// TIA Portal V16 export
// export: Created 2024-12-03T15:41:42.9786979Z, ExportSetting WithDefaults, DisplayName Totally Integrated Automation Portal, DisplayVersion V16 Update 6, DisplayName TIA Portal Version Control Interface, DisplayVersion V16 Update 2, DisplayName TIA Portal Openness, DisplayVersion V16 Update 6, DisplayName TIA Portal Teamcenter Gateway, DisplayVersion V16, DisplayName SINAMICS Startdrive Advanced, DisplayVersion V16 Update 5, DisplayName SINAMICS Startdrive G130, G150, S120, S150, SINAMICS MV, S210, DisplayVersion V16 Update 5, DisplayName SINAMICS Startdrive G110M, G120, G120C, G120D, G120P, G115D, DisplayVersion V16 Update 5, DisplayName STEP 7 Professional, DisplayVersion V16 Update 6, DisplayName STEP 7 Safety, DisplayVersion V16, DisplayName WinCC Advanced / Unified PC, DisplayVersion V16 Update 6
FUNCTION_BLOCK "ZPA_Controller"   // FB23, SCL
{ S7_Optimized_Access := 'TRUE' }
VERSION : 0.1
// stored: AutoNumber true, IsIECCheckEnabled false, IsRetainMemResEnabled false, MemoryReserve 100, SetENOAutomatically false, UDAEnableTagReadback false
   VAR_INPUT
      I_ConnectUpStream : Bool := TRUE;
      I_StartedAutoMode : Bool;
      I_UseEncoder : Bool := true;
      I_BuildName : Bool := true;
      I_UseExternalReset : Bool := TRUE;
   END_VAR
   VAR_IN_OUT
      IO_Upstream : "Conveyor_UDT";
      IO_DownStream : "Conveyor_UDT";
      IO_COnv : "Conveyor_UDT";
   END_VAR
   VAR
      cyclerun : "CycleRun";
      Alarm : "AlarmInfo_UDT";
      AlarmInfoValue : String;
      ConveyorMode : Int;
      StepNumber : DInt;
      PrevStepNumber : DInt;
      ObjectRequestedMemory : Bool;
      ObjectReceivedFromDownStream : Bool;
      Step_105_GapTimeOk : Bool;
      GapTimeTimer : "TON_Encoder_FB";
      SleepTimer { S7_SetPoint := 'True'} : "TON_Encoder_FB";
      ToCloseDetection { S7_SetPoint := 'True'} : "TON_Encoder_FB";
      ToLongDetectionEnd { S7_SetPoint := 'True'} : "TON_Encoder_FB";
      ToLongDetectionStart { S7_SetPoint := 'True'} : "TON_Encoder_FB";
      ToSmallDetection { S7_SetPoint := 'True'} : "TON_Encoder_FB";
      DownStreamIsRunning { S7_SetPoint := 'True'} : Bool;
      DownStreamRunningPredictor : Int;
      ObjectReceivedDuringSending : Bool;
      BlockedRetry : Int;
      InitializeInternal : Bool;
      diag : Struct
         TrackingLost : UInt;
      END_STRUCT;
      StartupDelay : TON_TIME;
      Step_Init_10 { S7_SetPoint := 'True'} : "StepperController_Encoder";
      Step_Send_WaitAccumulate_100 { S7_SetPoint := 'True'} : "StepperController_Encoder";
      Step_Send_WaitReceive_105 { S7_SetPoint := 'True'} : "StepperController_Encoder";
      Step_Send_Sending_110 { S7_SetPoint := 'True'} : "StepperController_Encoder";
      Step_Send_RunEmpty_120 { S7_SetPoint := 'True'} : "StepperController_Encoder";
      Step_Rec_Waiting_200 { S7_SetPoint := 'True'} : "StepperController";
      Step_Rec_Request_210 { S7_SetPoint := 'True'} : "StepperController_Encoder";
      Step_Rec_receivingTillEnd_215 { S7_SetPoint := 'True'} : "StepperController_Encoder";
      Step_Rec_RequetContiue_220 { S7_SetPoint := 'True'} : "StepperController_Encoder";
      Step_RequestObject_400_1 { S7_SetPoint := 'True'} : "StepperController_Encoder";
      Step_RequestObject_400_2 { S7_SetPoint := 'True'} : "StepperController_Encoder";
      Encoder { S7_SetPoint := 'True'} : "Virtual_Encoder_FB";
      BlockAlarmReceive { S7_SetPoint := 'True'} : Program_Alarm;
      BlockedSending { S7_SetPoint := 'True'} : Program_Alarm;
      ToCloseALarm { S7_SetPoint := 'True'} : Program_Alarm;
      ToSmallAlarm { S7_SetPoint := 'True'} : Program_Alarm;
      ToLongAlarm { S7_SetPoint := 'True'} : Program_Alarm;
      ResetMirror { S7_SetPoint := 'True'} : Bool;
   END_VAR
   VAR_TEMP
      T_ZoneInfo : "ZoneInfo";
      T_Appstate : "ApplicationState_UDT";
      T_Condition : Bool;
      T_Condtion_1 : Bool;
      T_Condtion_2 : Bool;
      T_NextStepNumber : DInt;
      T_TimeOutStepNumber : DInt;
      T_ConditionTime : Time;
      T_RunSent : Bool;
      T_RunReceive : Bool;
      T_RunInit : Bool;
      T_ReceiveTransferUnit : Bool;
      T_SleepMode : Bool;
      T_StandbyMode : Bool;
      T_Dummy : Bool;
   END_VAR
   VAR CONSTANT
      Step_TimeOutSending : DInt := 910;
      Step_TImeOutReceiving : DInt := 810;
      Step_ToCloseAlarm : DInt := 920;
      Step_ToSmall : DInt := 930;
      Step_ToLong : DInt := 940;
   END_VAR
BEGIN
   #T_ZoneInfo := "ApplicationState_DB".ZoneNames[#IO_COnv.Zone];
   #T_Appstate := "ApplicationState_DB".Appstate[#T_ZoneInfo.AppStateIndex];
   #ConveyorMode := #IO_COnv.Settings.Mode;

   IF "RunTime_DB".CycleRun = #T_ZoneInfo.AppStateIndex THEN
       #cyclerun();
   END_IF;

   #T_NextStepNumber := 0;
   #T_Condition := false;

   REGION ENCODER

       IF #I_UseEncoder THEN

           IF #IO_COnv.Cmd.RunAuto AND #IO_COnv.Input.Running_FB THEN
               #Encoder.I_CurrentRelativeSpeed_Perc := #IO_COnv.Cmd.SpeedAuto;
           ELSE
               #Encoder.I_CurrentRelativeSpeed_Perc := 0.0;
           END_IF;

           #Encoder(I_RelativeReferenceSpeed_Perc := #IO_COnv.Encoder.Settings.BaseRelative,
                    I_AbsoluteSpeedOnReferecne_m_min := #IO_COnv.Encoder.Settings.Base_M_min,
                    IO_VirtualEncoder := #IO_COnv.Encoder);

       END_IF;

   END_REGION

   REGION AUTO BUFFER MODE

       IF #IO_COnv.Settings.AutomaticBuffering
           AND #IO_COnv.Settings.Mode = "RUNTILLEND_MODE" THEN

           IF #ConveyorMode = "BUFFER_MODE" AND #IO_DownStream.Status.Empty THEN
               RESET_TIMER(#Step_Rec_Waiting_200.S_TimeOutTime);
           END_IF;

           IF #IO_DownStream.Status.Empty THEN
               #ConveyorMode := "RUNTILLEND_MODE";
           END_IF;

           IF NOT #IO_DownStream.Status.Empty AND NOT #IO_DownStream.Input.Running_FB AND #IO_DownStream.Input.SensorAtEndLogic.State THEN
               #ConveyorMode := "BUFFER_MODE";
           END_IF;

       END_IF;

   END_REGION

   REGION Init

       IF (NOT #T_Appstate.States.AutoModeActivated.State AND #StepNumber < 800) OR #StepNumber  = 0
           OR #IO_COnv.Status.ManualMode THEN
           #IO_COnv.Status.Initialized := FALSE;
           #StepNumber := -10;
           #IO_COnv.Status.StartedAutoMode := FALSE;
           #IO_COnv.Status.Empty := FALSE;
       END_IF;

       IF #IO_COnv.Cmd.ReInitialize OR #InitializeInternal
           OR ((#T_Appstate.Hmi_Buttons.reset.state.LE OR #IO_COnv.Cmd.Reset) AND #IO_COnv.Alarms.Status > 0) THEN

           #IO_COnv.Cmd.ReInitialize := FALSE;
           #IO_COnv.Status.Initialized := FALSE;
           #IO_COnv.Status.Empty := FALSE;
           #ObjectReceivedFromDownStream := FALSE;
           #StepNumber := 10;

           #ToCloseDetection.I_ResetHandshake := 1;
           #ToLongDetectionEnd.I_ResetHandshake := 1;
           #ToLongDetectionStart.I_ResetHandshake := 1;
           #ToSmallDetection.I_ResetHandshake := 1;

           IF NOT #InitializeInternal THEN
               #BlockedRetry := 0;
           END_IF;

           #InitializeInternal := FALSE;

       END_IF;

       IF #T_Appstate.States.AutoModeActivated.State
           AND NOT #IO_COnv.Status.ManualMode
           AND NOT #IO_COnv.Status.Initialized
           AND (#StepNumber = -10 OR #StepNumber = 0)
           AND (#IO_DownStream.Status.StartedAutoMode OR #I_StartedAutoMode)
       THEN
           #StepNumber := 10;
       END_IF;

       IF NOT #I_StartedAutoMode THEN
           #StartupDelay(IN := #T_Appstate.States.AutoModeActivated.State AND #IO_DownStream.Status.StartedAutoMode, //AND (NOT #IO_COnv.Alarms.MotorAlarm.Active OR #IO_COnv.Status.StartedAutoMode),
                         PT := #IO_COnv.Settings.Timings.StartupDelay,
                         Q => #IO_COnv.Status.StartedAutoMode);

       ELSE
           #IO_COnv.Status.StartedAutoMode := TRUE;
       END_IF;

       #Step_Init_10(I_StepNumber := 10,
                      I_NextStepNumber := 100,
                      I_TimeOutStepNumber := 200,
                      I_Condition := #IO_COnv.Input.SensorAtEndLogic.State,
                      I_TimeOutDistance := #IO_COnv.Settings.Timings.InitDistance,
                      I_PauseTimeOut := NOT #IO_COnv.Input.Running_FB,
                      I_AccumulateConditionTIme := TRUE,
                      I_DeltaDistance := #IO_COnv.Encoder.Distance_mm,
                      IO_PrevStepNumber := #PrevStepNumber,
                      IO_StepNumber := #StepNumber);

       IF #StepNumber <> -10 AND #StepNumber <> 10 THEN
           #IO_COnv.Status.Initialized := true;
       END_IF;

   END_REGION

   REGION STANDBY

       #T_StandbyMode := #T_Appstate.States.Standby.State AND NOT #IO_COnv.Cmd.IgnoreStandby;

   END_REGION

   REGION ACCUMULATION

       #IO_COnv.Status.AccumulationOn :=
       #IO_COnv.Cmd.Accumulate.Acc_ext_1 OR
       #IO_COnv.Cmd.Accumulate.Acc_ext_2 OR
       #IO_COnv.Cmd.Accumulate.Acc_ext_3 OR
       #IO_COnv.Cmd.Accumulate.Acc_ext_4 OR
       #IO_COnv.Cmd.Accumulate.Acc_ext_5 OR
       #IO_COnv.Cmd.Accumulate.Acc_Scale_1 OR
       #IO_COnv.Cmd.Accumulate.Acc_Scale_2 OR
       #IO_COnv.Cmd.Accumulate.Acc_Scale_3 OR
       #IO_COnv.Cmd.Accumulate.Acc_Scan_1 OR
       #IO_COnv.Cmd.Accumulate.Acc_Scan_2 OR
       #IO_COnv.Cmd.Accumulate.Acc_Scan_3 OR
       #IO_COnv.Cmd.Accumulate.Acc_TC_1 OR
       #IO_COnv.Cmd.Accumulate.Acc_TC_2 OR
       #IO_COnv.Cmd.Accumulate.Acc_TC_3;

   END_REGION

   REGION Conveyor emprty

       CASE #ConveyorMode OF
               "ZPA_TRAIN_MODE",
           "ZPA_MODE":
               #IO_COnv.Status.Empty := #IO_COnv.Status.Empty := #StepNumber = 200 AND NOT #IO_COnv.Input.SensorAtEndLogic.State;
           "RUNTILLEND_MODE":
               #IO_COnv.Status.Empty := #IO_COnv.Status.Empty := #StepNumber = 200 AND NOT #IO_COnv.Input.SensorAtEndLogic.State;
           "BUFFER_MODE":
               #IO_COnv.Status.Empty := FALSE;
       END_CASE;

   END_REGION

   REGION Running empty / request object

       //This function disables train mode because an object was requested
       IF #StepNumber = 200 OR #StepNumber = 0 OR #StepNumber = -10 THEN
           #ObjectRequestedMemory := false;
       END_IF;

       // IF #IO_COnv.Input.SensorAtStart.State OR #IO_COnv.Cmd.StartRequestObject THEN
       //     RESET_TIMER(#RequestObject_400_1.S_TimeOutTime);
       // END_IF;

       IF #IO_COnv.Cmd.StartRequestObject AND #StepNumber >= 200 AND #StepNumber <220 THEN
           #StepNumber := 400;
           #IO_COnv.Cmd.StartRequestObject := FALSE;
           #ObjectRequestedMemory := true;
       END_IF;

       #Step_RequestObject_400_1(I_StepNumber:=400,
                            I_NextStepNumber:=100,
                            I_TimeOutStepNumber:=200,
                            I_ErrorConditon := #IO_COnv.Cmd.StopRequestObject,
                            I_ErrorStepNumber := 200,
                            I_Condition:= #IO_COnv.Input.SensorAtEndLogic.State,
                            I_TimeOutDistance:=#IO_COnv.Settings.Timings.ConveyorLength,
                            I_PauseTimeOut:= NOT #IO_COnv.Input.Running_FB,
                            I_IgnoreTimeOut:=FALSE,
                            I_AccumulateConditionTIme:=TRUE,
                            I_DeltaDistance := #IO_COnv.Encoder.Distance_mm,
                            IO_PrevStepNumber := #PrevStepNumber,
                            IO_StepNumber:=#StepNumber);

   END_REGION

   REGION Receiving

       IF #StepNumber >= 200 AND #StepNumber < 215
           AND #StepNumber < 800
           AND #IO_COnv.Input.SensorAtEndLogic.State AND (#ConveyorMode = "ZPA_MODE" OR #ConveyorMode = "ZPA_TRAIN_MODE") THEN
           #StepNumber := 215;
       END_IF;

       REGION OBJECT RECEIVED DURING SENDING
           //IF #I_Upstream.Status.ObjectSentPulse
           IF #IO_COnv.Input.SensorAtStartLogic.LE
             //  AND #I_Upstream.Status.ObjectSentPulse
               AND #IO_COnv.Status.ExecutingSendingSequence
               AND #ConveyorMode = "ZPA_TRAIN_MODE" THEN
               #ObjectReceivedDuringSending := true;
           END_IF;
       END_REGION

       REGION STEP 200 WAIT FOR RECEIVING


           #T_Condition := #IO_Upstream.Cmd.ReadyToSent AND #I_ConnectUpStream;
           #Step_Rec_Waiting_200(I_StepNumber := 200,
                             I_TimeOutStepNumber := 200,
                             I_NextStepNumber := 210,
                             I_Condition := #T_Condition,
                             I_ConditionTIme := #IO_COnv.Settings.Timings.DelayedStart,
                             I_IgnoreTimeOut := TRUE,
                             IO_PrevStepNumber := #PrevStepNumber,
                             IO_StepNumber := #StepNumber);

       END_REGION

       REGION STEP 210 Object received

           IF #ConveyorMode = "ZPA_MODE"
               OR #ConveyorMode = "ZPA_TRAIN_MODE"
               OR #ConveyorMode = "BUFFER_MODE"
               OR #ConveyorMode = "RUNTILLEND_MODE" THEN
               #T_Condition := #IO_COnv.Input.SensorAtStartLogic.FE;
           END_IF;

           #Step_Rec_Request_210(I_StepNumber := 210,
                             I_NextStepNumber := 215,
                             I_TimeOutStepNumber := 200,
                             I_IgnoreTimeOut := FALSE,
                             I_TimeOutDistance := #IO_COnv.Settings.Timings.ConveyorLength,
                             I_PauseTimeOut := NOT #IO_COnv.Input.Running_FB AND #IO_Upstream.Cmd.ReadyToSent AND #IO_COnv.Input.SensorAtStartLogic.State,
                             I_Condition := #T_Condition,
                             I_DeltaDistance := #IO_COnv.Encoder.Distance_mm,
                             IO_PrevStepNumber := #PrevStepNumber,
                             IO_StepNumber := #StepNumber);

           REGION Skip receive till end (215) when in buffer mode
               IF #StepNumber = 215  AND #ConveyorMode = "BUFFER_MODE" THEN
                   #StepNumber := 220;
               END_IF;
           END_REGION

       END_REGION

       REGION STEP 215 RECVEIVE TILL END (alarm active)

           IF #ConveyorMode = "ZPA_MODE" OR #ConveyorMode = "RUNTILLEND_MODE"
               OR #ConveyorMode = "ZPA_TRAIN_MODE"
           THEN
               #T_Condition := #IO_COnv.Input.SensorAtEndLogic.State;
           END_IF;

           IF #IO_COnv.Settings.Alarms.BlockDetectionOn THEN
               #T_TimeOutStepNumber := #Step_TImeOutReceiving;
           ELSE
               #T_TimeOutStepNumber := 200;
           END_IF;

           #Step_Rec_receivingTillEnd_215(I_StepNumber := 215,
                                 I_NextStepNumber := 220,
                                 I_TimeOutStepNumber := #T_TimeOutStepNumber,
                                 I_IgnoreTimeOut := FALSE,
                                 I_TimeOutDistance := #IO_COnv.Settings.Timings.ConveyorLength,
                                 I_PauseTimeOut := NOT #IO_COnv.Input.Running_FB,
                                 I_Condition := #T_Condition,
                                 I_DeltaDistance := #IO_COnv.Encoder.Distance_mm,
                                 IO_PrevStepNumber := #PrevStepNumber,
                                 IO_StepNumber := #StepNumber);

           REGION ALARMS HANDELING

               IF #Step_Rec_receivingTillEnd_215.O_ConditionTrans THEN
                   #ObjectReceivedDuringSending := FALSE;
                   #BlockedRetry := 0;
               END_IF;

           END_REGION

       END_REGION

       REGION STEP 220 RECEIVE RUNNING HOLD ON

           IF #ConveyorMode = "ZPA_MODE" OR #ConveyorMode = "RUNTILLEND_MODE"
               OR #ConveyorMode = "ZPA_TRAIN_MODE"
           THEN
               #T_NextStepNumber := 100;
           END_IF;

           IF #ConveyorMode = "BUFFER_MODE" THEN
               #T_NextStepNumber := 200;
           END_IF;

           #Step_Rec_RequetContiue_220(I_StepNumber := 220,
                                   I_NextStepNumber := #T_NextStepNumber,
                                   I_Condition := #IO_COnv.Input.Running_FB,
                                   I_AccumulateConditionTIme := TRUE,
                                   I_ConditionDistance := #IO_COnv.Settings.Timings.ReceiveDistance,
                                   I_IgnoreTimeOut := TRUE,
                                   I_DeltaDistance := #IO_COnv.Encoder.Distance_mm,
                                   IO_PrevStepNumber := #PrevStepNumber,
                                   IO_StepNumber := #StepNumber);

           IF #Step_Rec_RequetContiue_220.O_ConditionTrans THEN
               #ObjectReceivedFromDownStream := TRUE;
           END_IF;

       END_REGION

       REGION GET NEW TRACKING

           REGION TRACK RECEIVING HANDLEING
               IF #ConveyorMode = "ZPA_TRAIN_MODE" OR #ConveyorMode = "ZPA_MODE" THEN
                   #IO_COnv.TrackingStat.TrackingReceived := FALSE;

                   // Clear currnet tracking if we are inducting the code
                   // If not this can cause timing issues
                   IF #IO_COnv.Status.ObjectOnConveyor AND #Step_Rec_Request_210.O_ConditionTrans THEN
                       #IO_COnv.TrackingStat.Current := "Tracking_DB".EmptyTrackingSimple;
                   END_IF;



                   // Receive upstream tracking
                   // Only do this if this is on a non inducting code point
                   IF NOT  #IO_COnv.Status.ObjectOnConveyor AND
                       #Step_Rec_receivingTillEnd_215.O_ConditionTrans AND NOT #IO_COnv.TrackingCmd.InductNewTracking THEN
                       #IO_COnv.TrackingStat.Current := #IO_Upstream.TrackingStat.InSending;
                       #IO_COnv.TrackingStat.TrackingReceived := TRUE;

                       // //Tracking diagnostics
                       // IF #IO_COnv.TrackingStat.Current.Barcode = '' OR #IO_COnv.TrackingStat.Current.PLC_Dest = 0 THEN
                       //     #IO_COnv.TrackingStat.Current.Barcode := 'TRACKING_LOST';
                       //     #IO_COnv.TrackingStat.Current.PLC_Dest := 99;
                       //     #diag.TrackingLost += 1;
                       // END_IF;

                   END_IF;
               END_IF;

           END_REGION

           IF #IO_COnv.TrackingCmd.InductNewTracking AND #IO_COnv.Status.ObjectOnConveyor THEN
               #IO_COnv.TrackingStat.Current := #IO_COnv.TrackingCmd.NewTrackingId;
               #IO_COnv.TrackingCmd.InductNewTracking := 0;
           END_IF;

       END_REGION

       IF NOT #IO_COnv.Input.SensorAtEndLogic.State THEN
           #ObjectReceivedFromDownStream := FALSE;
       END_IF;

   END_REGION

   REGION Sending

       //ZPA mode jump to receive 
       IF (#ConveyorMode = "ZPA_MODE" OR #ConveyorMode = "ZPA_TRAIN_MODE" OR #ConveyorMode = "RUNTILLEND_MODE")  AND #StepNumber = 100
           AND #StepNumber < 800
           AND NOT #IO_COnv.Input.SensorAtEndLogic.State THEN
           #StepNumber := 200;
       END_IF;

       //Buffer mode or run till end jump to sending when object at end
       IF (#ConveyorMode = "BUFFER_MODE" OR #ConveyorMode = "RUNTILLEND_MODE")
           AND #IO_COnv.Input.SensorAtEndLogic.State AND (#StepNumber < 100 OR #StepNumber >= 200) AND #StepNumber < 800 THEN
           #StepNumber := 220;
       END_IF;

       REGION STEP100 WIAT FOR NO ACCUMULATION AND START SNEDING PROCESS

           IF #ConveyorMode = "ZPA_MODE"
               OR #ConveyorMode = "ZPA_TRAIN_MODE"
               OR #ConveyorMode = "BUFFER_MODE"
               OR #ConveyorMode = "RUNTILLEND_MODE" THEN
               #T_Condition := NOT #IO_COnv.Status.AccumulationOn;
           END_IF;

           #Step_Send_WaitAccumulate_100(I_StepNumber := 100,
                                     I_NextStepNumber := 105,
                                     I_ConditionDistance := 0.0,
                                     I_Condition := #T_Condition
                                     AND NOT #T_StandbyMode,
                                     I_IgnoreTimeOut := TRUE,
                                     IO_PrevStepNumber := #PrevStepNumber,
                                     IO_StepNumber := #StepNumber);

           IF #Step_Send_WaitAccumulate_100.O_ConditionTrans THEN
               #ObjectReceivedFromDownStream := FALSE;
           END_IF;

       END_REGION

        REGION STEP105 WIAT for downstream is ready to receive

            REGION GAP TIME OK

                #GapTimeTimer(I_Start := #IO_DownStream.Input.Running_FB AND NOT #IO_COnv.Input.SensorAtEndLogic.FE,
                              I_Reset:= #IO_COnv.Input.SensorAtEndLogic.FE,
                              I_DeltaDistance_mm := #IO_DownStream.Encoder.Distance_mm,
                              I_SetPoint:= #IO_COnv.Settings.Timings.GapDistance,
                              I_Remanent := true,
                              Q => #Step_105_GapTimeOk);

                IF #IO_COnv.Settings.Timings.GapDistance = 0.0 THEN
                    #Step_105_GapTimeOk := true;
                END_IF;

            END_REGION

            IF #ConveyorMode = "ZPA_MODE"
                OR #ConveyorMode = "ZPA_TRAIN_MODE"
                OR #ConveyorMode = "BUFFER_MODE"
                OR #ConveyorMode = "RUNTILLEND_MODE" THEN
                #T_Condition := #IO_DownStream.Cmd.ReadyToReceive;
            END_IF;

            #Step_Send_WaitReceive_105(I_StepNumber := 105,
                                 I_NextStepNumber := 110,
                                 I_Condition := #T_Condition AND #Step_105_GapTimeOk,
                                 I_ConditionDistance := 0.0,
                                 I_AccumulateConditionTIme := true,
                                 I_IgnoreTimeOut := TRUE,
                                 IO_PrevStepNumber := #PrevStepNumber,
                                 IO_StepNumber := #StepNumber);

            #IO_COnv.Status.ObjectSentPulse := FALSE;
            IF #Step_Send_WaitReceive_105.O_ConditionTrans THEN
                #IO_COnv.Status.ObjectSentPulse := true;
            END_IF;

        END_REGION

        REGION STEP 110 SENT TILL NO SENSOR END PRESENT (ALARM ACTIVE)

            IF #ConveyorMode = "ZPA_MODE"
                OR #ConveyorMode = "ZPA_TRAIN_MODE"
                OR #ConveyorMode = "BUFFER_MODE"
                OR #ConveyorMode = "RUNTILLEND_MODE" THEN
                #T_Condition := NOT #IO_COnv.Input.SensorAtEndLogic.State;
           END_IF;

           IF #IO_COnv.Settings.Alarms.BlockDetectionOn THEN
               #T_TimeOutStepNumber := #Step_TimeOutSending;
           ELSE
               #T_TimeOutStepNumber := 200;
           END_IF;

           #Step_Send_Sending_110(I_StepNumber := 110,
                              I_NextStepNumber := 120,
                              I_TimeOutStepNumber := #T_TimeOutStepNumber,
                              I_IgnoreTimeOut := FALSE,
                              I_Condition := #T_Condition,
                              I_TimeOutDistance := #IO_COnv.Settings.Alarms.SentTimeError,
                              I_PauseTimeOut := NOT #IO_COnv.Input.Running_FB,
                              I_DeltaDistance := #IO_COnv.Encoder.Distance_mm,
                              IO_PrevStepNumber := #PrevStepNumber,
                              IO_StepNumber := #StepNumber);

           REGION ALARMS HANDELING

               IF #Step_Send_Sending_110.O_ConditionTrans THEN
                   #BlockedRetry := 0;
               END_IF;

           END_REGION

       END_REGION

       REGION STEP 120 SENT RUN WITH A HOLD ON TIME

           IF #ConveyorMode = "ZPA_TRAIN_MODE" THEN
               IF #ObjectReceivedDuringSending THEN
                   #Step_Rec_receivingTillEnd_215.TimeOutTime.I_ResetHandshake := true;
                   #T_NextStepNumber := 210;
               ELSE
                   #T_NextStepNumber := 200;
               END_IF;
           ELSE
               #T_NextStepNumber := 200;
           END_IF;

           #Step_Send_RunEmpty_120(I_StepNumber := 120,
                               I_NextStepNumber := #T_NextStepNumber,
                               I_Condition := #IO_COnv.Input.Running_FB,
                               I_IgnoreTimeOut := TRUE,
                               I_ConditionDistance := #IO_COnv.Settings.Timings.SendDistance,
                               I_AccumulateConditionTIme := TRUE,
                               I_DeltaDistance := #IO_COnv.Encoder.Distance_mm,
                               IO_PrevStepNumber := #PrevStepNumber,
                               IO_StepNumber := #StepNumber);

       END_REGION

       REGION SET NEW TRAKCING IN SENDING

           // IF #ConveyorMode = "ZPA_TRAIN_MODE" OR #ConveyorMode = "ZPA_MODE" THEN
           //     IF #Step_Send_WaitReceive_105.O_ConditionTrans THEN
           //         #IO_COnv.TrackingStat.InSending := #IO_COnv.TrackingStat.Current;
           //     END_IF;
           // END_IF;
           // 

           #T_Condition := #ConveyorMode = "ZPA_TRAIN_MODE" OR #ConveyorMode = "ZPA_MODE";
           #T_Condition := #T_Condition AND NOT #IO_COnv.TrackingCmd.InductNewTracking;

           #T_Condtion_1 := #T_Condition AND  ((#StepNumber = 100 OR #StepNumber = 105) AND #IO_DownStream.Status.Empty);
           #T_Condtion_2 := #T_Condition AND #Step_Send_WaitReceive_105.O_ConditionTrans;

           IF #T_Condtion_1 OR #T_Condtion_2 THEN
               #IO_COnv.TrackingStat.InSending := #IO_COnv.TrackingStat.Current;
           END_IF;

       END_REGION

   END_REGION

   REGION Reset stepnumber AND status when object is removed AND conveyor was NOT running

       IF #IO_COnv.Input.SensorAtEndLogic.FE
           AND #IO_COnv.Settings.AutoReset
           AND #StepNumber >= 100
           AND #StepNumber < 800
           AND NOT #IO_COnv.Cmd.RunAuto THEN
           // #IO_COnv.TrackingCmd.ClearTracking := TRUE;
           #StepNumber := 200;
           //#StepNumber := 8000;
       END_IF;

   END_REGION

   REGION CLEAR TRACKING

       // IF #IO_DownStream.TrackingStat.TrackingReceived THEN
       //     #IO_COnv.TrackingStat.InSending := "Tracking_DB".EmptyTrackingSimple;
       // END_IF;

       #IO_COnv.TrackingStat.TrackingCleared := FALSE; //Tracking cleared status is only one cycle high

       IF (#IO_DownStream.TrackingStat.TrackingReceived AND #ConveyorMode = "ZPA_MODE")
           OR (#IO_COnv.Input.SensorAtEndLogic.FE AND (#ConveyorMode = "ZPA_TRAIN_MODE" OR #ConveyorMode = "ZPA_MODE"))
           OR #IO_COnv.TrackingCmd.ClearTracking THEN
           //#IO_COnv.TrackingStat.Current := "Tracking_DB".EmptyTrackingSimple;
           //#IO_COnv.TrackingStat.InSending := "Tracking_DB".EmptyTrackingSimple;
           #IO_COnv.TrackingStat.TrackingCleared := TRUE;
           #IO_COnv.TrackingCmd.ClearTracking := FALSE;
       END_IF;

   END_REGION

   REGION DOWNSTREAM RUNNING

       IF #DownStreamRunningPredictor <= 4 THEN
           #DownStreamRunningPredictor += 1;
       END_IF;

       IF NOT #IO_DownStream.Input.Running_FB THEN
           #DownStreamIsRunning := false;
       END_IF;

       IF #DownStreamRunningPredictor > 4 THEN
           #DownStreamIsRunning := FALSE;
       END_IF;

       IF #Step_Send_WaitReceive_105.O_ConditionTrans OR #IO_DownStream.Input.Running_FB THEN
           #DownStreamRunningPredictor := 0;
       END_IF;

       IF #IO_DownStream.Input.Running_FB OR #DownStreamRunningPredictor < 4 THEN
           #DownStreamIsRunning := true;
       END_IF;


   END_REGION

   REGION SLEEPTIMER

       #T_Condition :=
       #IO_Upstream.Status.ExecutingReceiveSequence
       OR #IO_Upstream.Status.RequestForSending
       OR #IO_Upstream.Status.ExecutingSendingSequence;

       #T_Condition := #T_Condition AND #I_ConnectUpStream;

       IF #T_Condition
           OR #Step_Rec_Request_210.O_ConditionTrans
       THEN
           #SleepTimer.I_ResetHandshake := true;
       END_IF;

       #T_Condition := NOT #IO_COnv.Status.ExecutingSendingSequence
       AND NOT #IO_COnv.Status.RequestForSending
       AND NOT #ObjectRequestedMemory
       AND NOT #IO_COnv.Status.ExecutingReceiveSequence
       AND NOT #IO_COnv.Cmd.ManualOverride
       AND #T_Appstate.States.AutoModeActivated.State
       AND NOT #IO_COnv.Cmd.Reset
       AND NOT #IO_COnv.Input.SensorAtStartLogic.State
       AND NOT #IO_COnv.Input.SensorAtEndLogic.State;

       #IO_COnv.Settings.Timings.SleepDistance := #IO_COnv.Settings.Timings.ConveyorLength;

       #SleepTimer(I_Start := #T_Condition,
                   I_SetPoint := #IO_COnv.Settings.Timings.SleepDistance,
                   I_DeltaDistance_mm := #IO_COnv.Encoder.Distance_mm);

       #T_SleepMode := #SleepTimer.Q AND #IO_COnv.Settings.EnergySave;

   END_REGION

   REGION ALARMS

       IF NOT #Alarm.init OR #IO_COnv.Name = '' OR #Alarm.info = '' OR "HMI_DB".ReloadSettings.signal THEN
           IF #I_BuildName THEN
               #IO_COnv.Name := "buildObjectName"(I_Symbolname := GetSymbolName(variable := #IO_COnv, size := 100));
               #Alarm.info := "buildAlarmInfo"(I_ObjectName := #IO_COnv.Name, I_ZoneIndex := #IO_COnv.Zone, I_ZoneName := #T_ZoneInfo.ZoneName);
               #Alarm.init := true;
           END_IF;
       END_IF;

       REGION DECIDE TO THROW BLOCK ALARM
           IF #StepNumber = #Step_TImeOutReceiving OR #StepNumber = #Step_TimeOutSending
               AND #BlockedRetry < #IO_COnv.Settings.Alarms.BlockRetrys THEN
               #BlockedRetry += 1;

               IF #BlockedRetry <= #IO_COnv.Settings.Alarms.BlockRetrys THEN
                   #InitializeInternal := true;
                   #StepNumber := 0;
               END_IF;

           END_IF;
       END_REGION

       REGION BLOCKED RECEIVE

           #IO_COnv.Alarms.BlockedReceive.Active := #StepNumber = #Step_TImeOutReceiving;
                   #IO_COnv.Alarms.Status.%X0 := #IO_COnv.Alarms.BlockedReceive.Active;

                   IF #cyclerun.O_Cycle = 1 AND "RunTime_DB".CycleRun = #T_ZoneInfo.AppStateIndex THEN
                       #BlockAlarmReceive(SIG := #IO_COnv.Alarms.BlockedReceive.Active,
                                          SD_1 := #Alarm.info,
                                          SD_2 := #T_ZoneInfo.ZoneName,
                                          SD_3 := #IO_COnv.Name);
                   END_IF;
       END_REGION

       REGION BLOCKED SENDING

           #IO_COnv.Alarms.BlockedSending.Active :=  #StepNumber = #Step_TimeOutSending;
                   #IO_COnv.Alarms.Status.%X1 := #IO_COnv.Alarms.BlockedSending.Active;

                   IF #cyclerun.O_Cycle = 2 AND "RunTime_DB".CycleRun = #T_ZoneInfo.AppStateIndex THEN
                       #BlockedSending(SIG := #IO_COnv.Alarms.BlockedSending.Active,
                                          SD_1 := #Alarm.info,
                                          SD_2 := #T_ZoneInfo.ZoneName,
                                          SD_3 := #IO_COnv.Name);
                   END_IF;
       END_REGION

       REGION TO CLOSE ALARM

           #ToCloseDetection(I_Start := NOT #IO_COnv.Input.SensorAtEndLogic.State AND #IO_COnv.Input.Running_FB,
                             I_Reset:= #IO_COnv.Input.SensorAtEndLogic.FE,
                             I_SetPoint:= #IO_COnv.Settings.Alarms.TimeBetweenParcels,
                             I_DeltaDistance_mm := #IO_COnv.Encoder.Distance_mm,
                             I_Remanent := true,
                             Q => #T_Dummy);

           IF NOT #ToCloseDetection.Q
               AND #IO_COnv.Input.SensorAtEndLogic.LE
               AND #IO_COnv.Cmd.RunAuto
               AND #IO_COnv.Settings.Alarms.ParcelsToCloseDetectionOn THEN
               #StepNumber := #Step_ToCloseAlarm;
           END_IF;

           #IO_COnv.Alarms.ToClose.Active := #StepNumber = #Step_ToCloseAlarm;
           #IO_COnv.Alarms.Status.%X3 := #IO_COnv.Alarms.ToClose.Active;

           IF #cyclerun.O_Cycle = 3 AND "RunTime_DB".CycleRun = #T_ZoneInfo.AppStateIndex THEN
               #ToCloseALarm(SIG := #IO_COnv.Alarms.ToClose.Active,
                             SD_1 := #Alarm.info,
                             SD_2 := #T_ZoneInfo.ZoneName,
                             SD_3 := #IO_COnv.Name);

           END_IF;

       END_REGION

       REGION TO SMALL ALAARM

           IF #IO_COnv.Input.SensorAtEndLogic.FE AND #IO_COnv.Cmd.RunAuto
               AND #IO_COnv.Settings.Alarms.ParcelToShortDetectionOn
               AND NOT #ToSmallDetection.Q THEN
               #StepNumber := #Step_ToSmall;
           END_IF;

           #ToSmallDetection(I_Start:=#IO_COnv.Input.SensorAtEndLogic.State AND #IO_COnv.Input.Running_FB,
                             I_Reset:= #IO_COnv.Input.SensorAtEndLogic.FE,
                             I_SetPoint:=#IO_COnv.Settings.Alarms.MinSizeParcel,
                             I_DeltaDistance_mm := #IO_COnv.Encoder.Distance_mm,
                             I_Remanent := true,
                             Q => #T_Dummy);

           #IO_COnv.Alarms.ToSmall.Active := #StepNumber = #Step_ToSmall;
           #IO_COnv.Alarms.Status.%X4 := #IO_COnv.Alarms.ToSmall.Active;

           IF #cyclerun.O_Cycle = 4 AND "RunTime_DB".CycleRun = #T_ZoneInfo.AppStateIndex THEN
               #ToCloseALarm(SIG := #IO_COnv.Alarms.ToSmall.Active,
                             SD_1 := #Alarm.info,
                             SD_2 := #T_ZoneInfo.ZoneName,
                             SD_3 := #IO_COnv.Name);
           END_IF;

       END_REGION

      REGION TO LONG ALARM

          // #T_Condition := #IO_COnv.Input.SensorAtStartLogic.State
          // AND #IO_COnv.Input.Running_FB
          // AND #I_Upstream.Input.Running_FB
          // AND #IO_COnv.Settings.Alarms.ParcelsToLongDetectionOn;

          #T_Condition :=
          (#IO_COnv.Input.Running_FB AND #IO_COnv.Input.SensorAtEndLogic.State AND #IO_COnv.Settings.Alarms.ParcelsToLongDetectionOn);

          #ToLongDetectionEnd(I_Start := #T_Condition,
                              I_Reset := #IO_COnv.Input.SensorAtEndLogic.LE OR #IO_COnv.Input.SensorAtEndLogic.FE,
                           I_SetPoint := #IO_COnv.Settings.Alarms.MaxSizeParcel * 4,
                           I_DeltaDistance_mm := #IO_COnv.Encoder.Distance_mm,
                           I_Remanent := true,
                           Q => #T_Dummy);

           #T_Condition :=
           (#IO_COnv.Input.Running_FB AND #IO_COnv.Input.SensorAtStartLogic.State AND #IO_COnv.Settings.Alarms.BlockedAtStartSensor);

          #ToLongDetectionStart(I_Start := #T_Condition,
                                I_Reset := #IO_COnv.Input.SensorAtStartLogic.LE OR #IO_COnv.Input.SensorAtStartLogic.FE,
                           I_SetPoint := #IO_COnv.Settings.Alarms.MaxSizeParcel * 4,
                           I_DeltaDistance_mm := #IO_COnv.Encoder.Distance_mm,
                           I_Remanent := true,
                           Q => #T_Dummy);

          IF #ToLongDetectionEnd.Q OR #ToLongDetectionStart.Q THEN
              #StepNumber := #Step_ToLong;
          END_IF;

          #IO_COnv.Alarms.ToLong.Active := #StepNumber = #Step_ToLong;
          #IO_COnv.Alarms.Status.%X5 := #IO_COnv.Alarms.ToLong.Active;

          IF #cyclerun.O_Cycle = 5 AND "RunTime_DB".CycleRun = #T_ZoneInfo.AppStateIndex THEN

              #ToLongAlarm(SIG := #IO_COnv.Alarms.ToLong.Active,
                           SD_1 := #Alarm.info,
                           SD_2 := #T_ZoneInfo.ZoneName,
                           SD_3 := #IO_COnv.Name);

          END_IF;

      END_REGION

      REGION MOTOR ALARM
          #IO_COnv.Alarms.Status.%X6 := #IO_COnv.Alarms.MotorAlarm.Active;
      END_REGION

      REGION BUNDLE ALARMS ACTIVE
          #IO_COnv.Alarms.AlarmActive.Active := #IO_COnv.Alarms.Status > 0;

          IF #IO_COnv.Alarms.Status > 0 THEN
              "ApplicationState_DB".Appstate[#T_ZoneInfo.AppStateIndex].Alarms.AlarmActiveInternalPLC := TRUE;
          END_IF;

      END_REGION

      REGION INIT AGAIN WHEN IN ALARM + RESET

          IF #IO_COnv.Alarms.Status > 0 AND ((#T_Appstate.Hmi_Buttons.reset.state.LE AND #I_UseExternalReset)
              OR #IO_COnv.Cmd.Reset) THEN
              #IO_COnv.Cmd.ReInitialize := true;
          END_IF;

          // IF #IO_COnv.Alarms.BlockedReceive.Active AND ((#T_Appstate.Hmi_Buttons.reset.state.LE AND #I_UseExternalReset)
          //     OR #IO_COnv.Cmd.Reset)
          // THEN
          //     #StepNumber := #PrevStepNumber;
          //     #BlockedRetry := 0;
          // END_IF;
      END_REGION

   END_REGION

   REGION Ready TO sent / receive

       //Init run commands
       #IO_COnv.Cmd.ReadyToSent := FALSE;
       #IO_COnv.Cmd.ReadyToSent := FALSE;
       #IO_COnv.Cmd.RunAuto := FALSE;
       #T_RunReceive := FALSE;
       #T_RunSent := FALSE;
       #T_RunInit := FALSE;

       REGION ZPA MODe sent receive
           IF #ConveyorMode = "ZPA_MODE" THEN

               #IO_COnv.Cmd.ReadyToSent := #StepNumber = 105 OR #StepNumber = 110 OR #StepNumber = 120;

               #IO_COnv.Cmd.ReadyToReceive := (#StepNumber = 200 OR #StepNumber = 210 OR #StepNumber = 400) AND NOT #IO_COnv.Input.SensorAtEndLogic.State;

               #T_RunInit := #StepNumber = 10 OR #StepNumber = 400;

               #T_RunReceive := #StepNumber = 200 AND #IO_COnv.Settings.RunIddle AND NOT #T_SleepMode
               AND NOT #T_StandbyMode;

               #T_RunReceive := #T_RunReceive OR #StepNumber = 210; //AND #IO_Upstream.Cmd.ReadyToSent;
               #T_RunReceive := #T_RunReceive OR #StepNumber = 215;
               #T_RunReceive := #T_RunReceive AND NOT #IO_COnv.Input.SensorAtEndLogic.State;
               #T_RunReceive := #T_RunReceive OR #StepNumber = 220;

               #T_RunSent := (#StepNumber = 110 AND #DownStreamIsRunning AND #IO_DownStream.Cmd.ReadyToReceive);

               IF #IO_COnv.Settings.SentHoldOnCheckReceive THEN
                   #T_RunSent := #T_RunSent OR (#StepNumber = 120 AND #IO_DownStream.Cmd.ReadyToReceive AND #DownStreamIsRunning);
               ELSE
                   #T_RunSent := #T_RunSent OR #StepNumber = 120;
               END_IF;

               #IO_COnv.Cmd.RunAuto := #T_RunInit OR #T_RunReceive OR #T_RunSent;
           END_IF;

       END_REGION

       REGION Runn till end sent receive

           IF #ConveyorMode = "RUNTILLEND_MODE" THEN

               #IO_COnv.Cmd.ReadyToSent := #StepNumber = 105 OR #StepNumber = 110 OR #StepNumber = 120;

               #IO_COnv.Cmd.ReadyToReceive := (#StepNumber = 200 OR #StepNumber = 210 OR #StepNumber = 215 OR #StepNumber = 220 OR #StepNumber = 400);
               #IO_COnv.Cmd.ReadyToReceive := #IO_COnv.Cmd.ReadyToReceive OR (#IO_COnv.Status.ExecutingSendingSequence AND  #IO_COnv.Input.Running_FB);

               #T_RunInit := #StepNumber = 10 OR #StepNumber = 400;

               #T_RunReceive := #StepNumber = 200 AND #IO_COnv.Settings.RunIddle
               AND NOT #T_SleepMode
               AND NOT #T_StandbyMode;
               #T_RunReceive := #T_RunReceive OR #StepNumber = 210;
               #T_RunReceive := #T_RunReceive OR #StepNumber = 215;
               #T_RunReceive := #T_RunReceive AND NOT #IO_COnv.Input.SensorAtEndLogic.State;
               #T_RunReceive := #T_RunReceive OR #StepNumber = 220;

               #T_RunSent := (#StepNumber = 110 AND #DownStreamIsRunning AND #IO_DownStream.Cmd.ReadyToReceive);

               IF #IO_COnv.Settings.SentHoldOnCheckReceive THEN
                   #T_RunSent := #T_RunSent OR (#StepNumber = 120 AND #IO_DownStream.Cmd.ReadyToReceive AND #DownStreamIsRunning);
               ELSE
                   #T_RunSent := #T_RunSent OR #StepNumber = 120 ;
               END_IF;

               #IO_COnv.Cmd.RunAuto := #T_RunInit OR #T_RunReceive OR #T_RunSent;
               #IO_COnv.Cmd.RunAuto := #IO_COnv.Cmd.RunAuto AND NOT #T_StandbyMode;
           END_IF;

       END_REGION

       REGION Buffer MODe sent receive
           IF #ConveyorMode = "BUFFER_MODE" THEN

               #IO_COnv.Cmd.ReadyToSent := #StepNumber = 105 OR #StepNumber = 110 OR #StepNumber = 120;

               #IO_COnv.Cmd.ReadyToReceive := (#StepNumber = 200 OR #StepNumber = 210 OR #StepNumber = 400);
               #IO_COnv.Cmd.ReadyToReceive := #IO_COnv.Cmd.ReadyToReceive OR (#IO_COnv.Cmd.ReadyToSent AND #IO_COnv.Cmd.RunAuto);

               #T_RunInit := #StepNumber = 10 OR #StepNumber = 400;

               #T_RunReceive := #StepNumber = 210 AND #IO_Upstream.Cmd.ReadyToSent;
               #T_RunReceive := #T_RunReceive OR #StepNumber = 215;
               #T_RunReceive := #T_RunReceive AND NOT #IO_COnv.Input.SensorAtEndLogic.State;
               #T_RunReceive := #T_RunReceive OR #StepNumber = 220;

               #T_RunSent := (#StepNumber = 110 AND #DownStreamIsRunning AND #IO_DownStream.Cmd.ReadyToReceive);

               IF #IO_COnv.Settings.SentHoldOnCheckReceive THEN
                   #T_RunSent := #T_RunSent OR (#StepNumber = 120 AND #IO_DownStream.Cmd.ReadyToReceive AND #DownStreamIsRunning);
               ELSE
                   #T_RunSent := #T_RunSent OR #StepNumber = 120;
               END_IF;

               #IO_COnv.Cmd.RunAuto := #T_RunInit OR #T_RunReceive OR #T_RunSent;
           END_IF;
       END_REGION

       REGION Train MODe sent receive

       END_REGION

       REGION ZPA TRAIN MODE
           IF #ConveyorMode = "ZPA_TRAIN_MODE" THEN

               #IO_COnv.Cmd.ReadyToSent := #StepNumber = 105 OR #StepNumber = 110 OR #StepNumber = 120;

               #IO_COnv.Cmd.ReadyToReceive := (#StepNumber = 200 OR #StepNumber = 210 OR #StepNumber = 400) AND NOT #IO_COnv.Input.SensorAtEndLogic.State;
               #IO_COnv.Cmd.ReadyToReceive := #IO_COnv.Cmd.ReadyToReceive
               OR (
               #IO_COnv.Status.ExecutingSendingSequence
               AND #IO_COnv.Cmd.RunAuto
               );

               #T_RunInit := #StepNumber = 10 OR #StepNumber = 400;

               #T_RunReceive := #StepNumber = 200 AND #IO_COnv.Settings.RunIddle AND NOT #T_SleepMode
               AND NOT #T_StandbyMode;
               #T_RunReceive := #T_RunReceive OR #StepNumber = 210; //AND (#I_Upstream.Cmd.ReadyToSent OR #ObjectReceivedDuringSending);
               #T_RunReceive := #T_RunReceive OR #StepNumber = 215;
               #T_RunReceive := #T_RunReceive AND NOT #IO_COnv.Input.SensorAtEndLogic.State;
               #T_RunReceive := #T_RunReceive OR #StepNumber = 220;

               #T_RunSent := (#StepNumber = 110 AND #DownStreamIsRunning AND #IO_DownStream.Cmd.ReadyToReceive);

               IF #IO_COnv.Settings.SentHoldOnCheckReceive THEN
                   #T_RunSent := #T_RunSent OR (#StepNumber = 120 AND #IO_DownStream.Cmd.ReadyToReceive AND #DownStreamIsRunning);
               ELSE
                   #T_RunSent := #T_RunSent OR #StepNumber = 120;
               END_IF;

               REGION FAST MODE
                   #IO_COnv.Cmd.ReadyToReceive := #IO_COnv.Cmd.ReadyToReceive
                   OR (
                   #IO_COnv.Status.ExecutingSendingSequence
                   AND #T_RunSent
                   );
               END_REGION

               #IO_COnv.Cmd.RunAuto := #T_RunInit OR #T_RunReceive OR #T_RunSent;
           END_IF;
       END_REGION

   END_REGION

   REGION Run motor

       #IO_COnv.Cmd.RunAuto := #IO_COnv.Cmd.RunAuto AND NOT #IO_COnv.Cmd.Interlock;

   END_REGION

   REGION Speed controller

       #IO_COnv.Cmd.SpeedAuto := #IO_COnv.Settings.Speed.speed;

       IF #IO_COnv.Settings.Speed.speedController THEN
           IF #IO_COnv.Input.SensorAtEndLogic.State
               AND #IO_DownStream.Cmd.RunAuto THEN
               #IO_COnv.Cmd.SpeedAuto := #IO_DownStream.Cmd.SpeedAuto * #IO_COnv.Settings.Speed.UpstreamGain;
           END_IF;
       END_IF;

   END_REGION

   REGION Create status

       //#IO_COnv.Status.ObjectOnConveyor := #StepNumber > 215 AND #StepNumber < 120;

       #IO_COnv.Status.ExecutingReceiveSequence := #StepNumber > 200 AND #StepNumber <= 220 OR #StepNumber = 400;
       #IO_COnv.Status.ExecutingSendingSequence := #StepNumber > 100 AND #StepNumber <= 120;
       #IO_COnv.Status.RequestForSending := (#StepNumber = 100 AND NOT #T_StandbyMode)
       OR #StepNumber = 105 OR #StepNumber = 110;

       #IO_COnv.Status.GapTimeOk := #Step_105_GapTimeOk;

   END_REGION

   REGION MANUAL MOTOR CONTROL

       #IO_COnv.Status.ManualMode := #T_Appstate.States.ManualModeActivated.State
       OR #IO_COnv.Cmd.ManualOverride;

       IF #IO_COnv.Cmd.ManualOverride THEN
           "ApplicationState_DB".Appstate[#T_ZoneInfo.AppStateIndex].States.ManaulOverrideActive.Internal := true;
       END_IF;

       IF "HMI_DB".RemoveManualOverride.signal
           OR NOT #T_Appstate.States.EmergencyOk.State THEN
           #IO_COnv.Cmd.ManualOverride := 0;
       END_IF;

       IF NOT #IO_COnv.Status.ManualMode THEN
           #IO_COnv.Cmd.RunManual := 0;
           #IO_COnv.Cmd.SpeedManual := 20.0;
       END_IF;

   END_REGION

   REGION INTERNAL RESET

       IF #ResetMirror THEN
           #IO_COnv.Cmd.Reset := 0;
       END_IF;

       #ResetMirror := #IO_COnv.Cmd.Reset;

   END_REGION
END_FUNCTION_BLOCK
